(* PLC project MotionTest1, Higen MCL 1 *)
(* stored: creationDateTime 2012-01-06T15:20:13, modificationDateTime 2026-03-05T12:13:42 *)

FUNCTION_BLOCK BlendTest
  VAR
    moveA : MC_MoveAbsolute;
    switch : MC_Power;
    readpos : MC_ReadActualPosition;
    setpos : MC_SetPosition;
    Block1 : MC_MoveAbsolute;
    readspeed : MC_ReadParameter;
  END_VAR
  VAR_INPUT
    Axis : AXIS_REF;
    Enable : BOOL;
    BlendMode : MC_BUFFER_MODE;
  END_VAR
  VAR_OUTPUT
    Done : BOOL;
    Pn : LREAL;
    Vn : LREAL;
  END_VAR

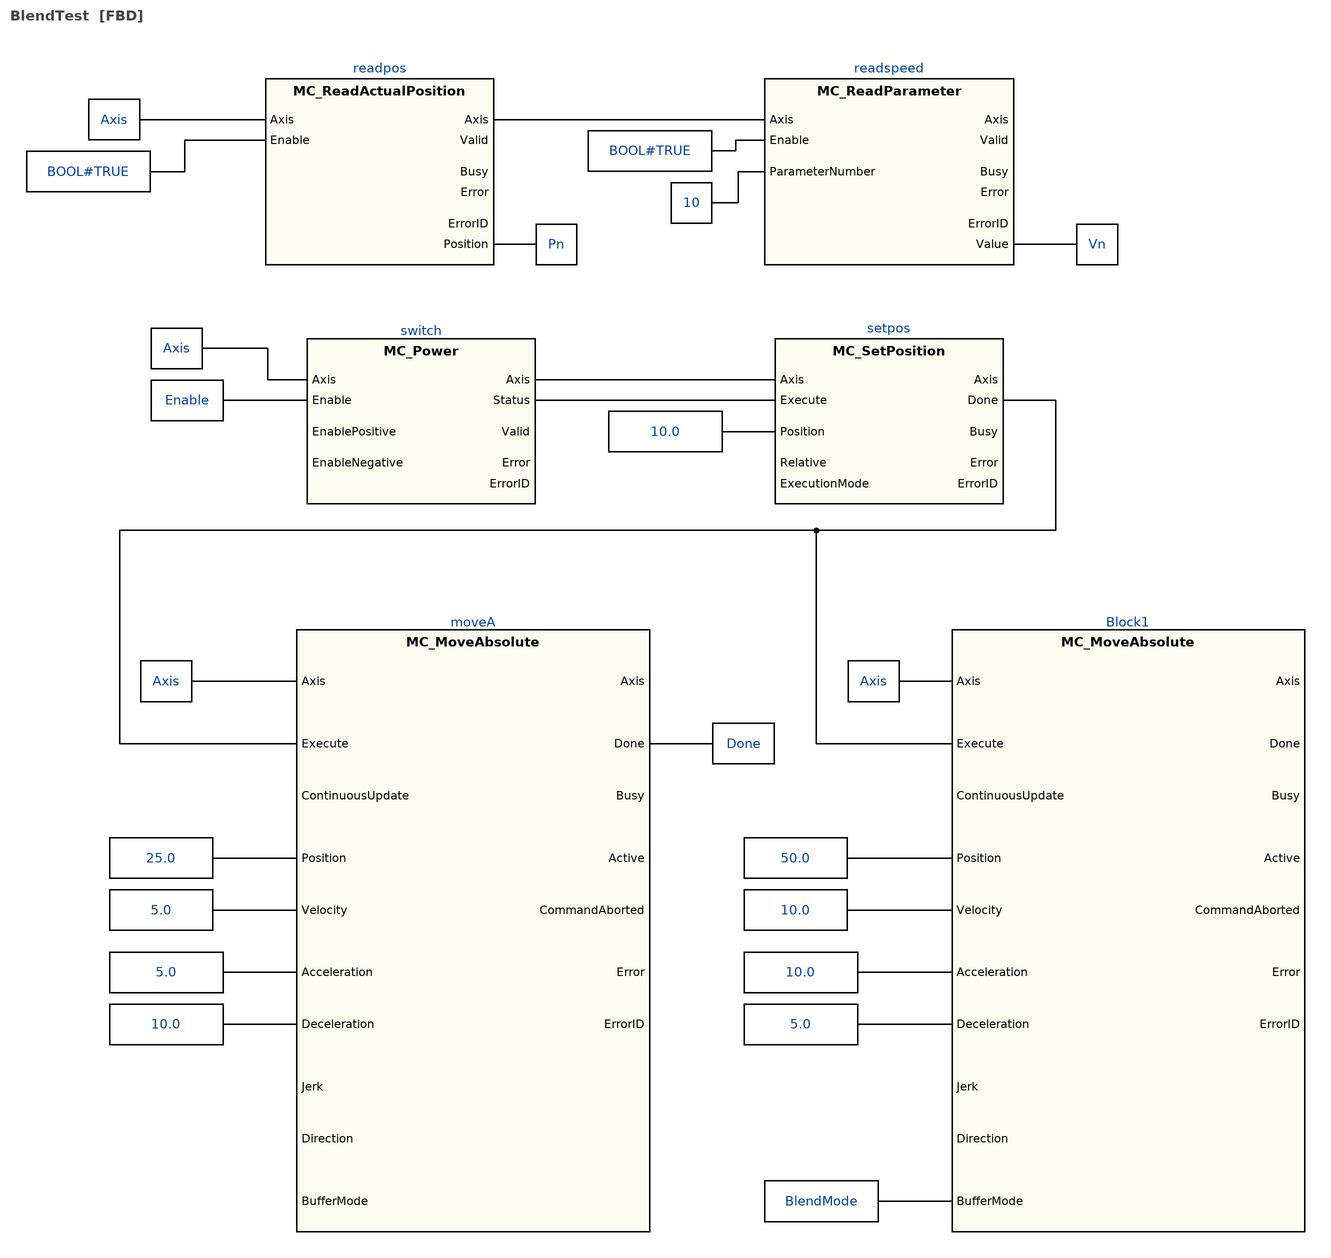
(* FBD diagram, written out as Structured Text *)
readpos(Axis := Axis, Enable := BOOL#TRUE);
Pn := readpos.Position;
switch(Axis := Axis, Enable := Enable);
setpos(Axis := switch.Axis, Execute := switch.Status, Position := 10.0);
moveA(Axis := Axis, Execute := setpos.Done, Position := 25.0, Velocity := 5.0, Acceleration := 5.0, Deceleration := 10.0);
Done := moveA.Done;
readspeed(Axis := readpos.Axis, Enable := BOOL#TRUE, ParameterNumber := 10);
Vn := readspeed.Value;
Block1(Axis := Axis, Execute := setpos.Done, Position := 50.0, Velocity := 10.0, Acceleration := 10.0, Deceleration := 5.0, BufferMode := BlendMode);
END_FUNCTION_BLOCK

PROGRAM main
  VAR
    clock : ULINT;
    High : BlendTest;
    Low : BlendTest;
    Previous : BlendTest;
    Next : BlendTest;
    r1 : R_TRIG;
    Block1 : R_TRIG;
    Block2 : R_TRIG;
    Block3 : R_TRIG;
    Block4 : BlendTest;
    Block5 : R_TRIG;
    sim0 : MC_Sim;
    sim1 : MC_Sim;
    sim2 : MC_Sim;
    sim3 : MC_Sim;
    sim4 : MC_Sim;
  END_VAR
  VAR  (* added by the conversion: wires and edge detectors of the diagram *)
    _SEL45_OUT : ANY;
    _SEL11_OUT : ANY;
    _SEL13_OUT : ANY;
    _SEL16_OUT : ANY;
    _SEL22_OUT : ANY;
  END_VAR

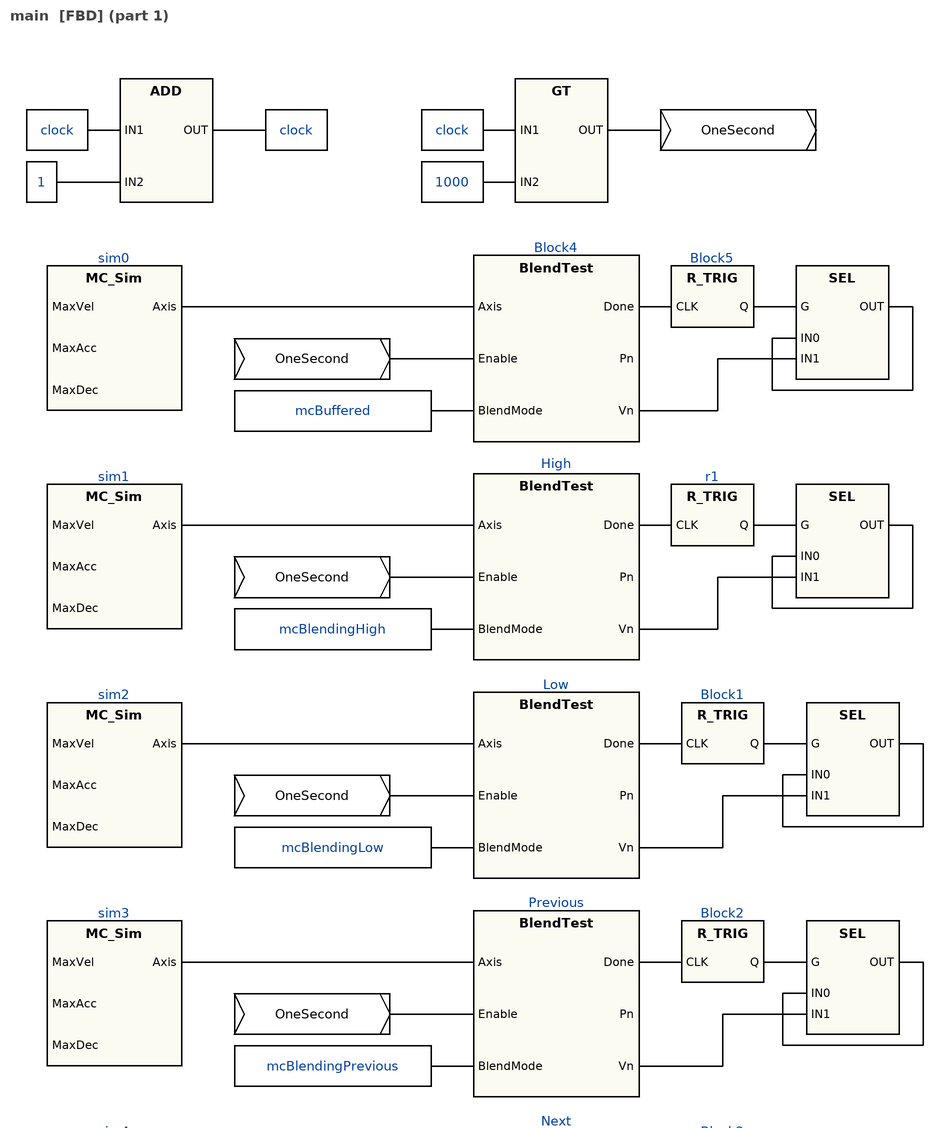
(* FBD diagram, written out as Structured Text *)
clock := clock + 1;
sim1();
High(Axis := sim1.Axis, Enable := clock > 1000, BlendMode := mcBlendingHigh);
sim2();
Low(Axis := sim2.Axis, Enable := clock > 1000, BlendMode := mcBlendingLow);
sim3();
Previous(Axis := sim3.Axis, Enable := clock > 1000, BlendMode := mcBlendingPrevious);
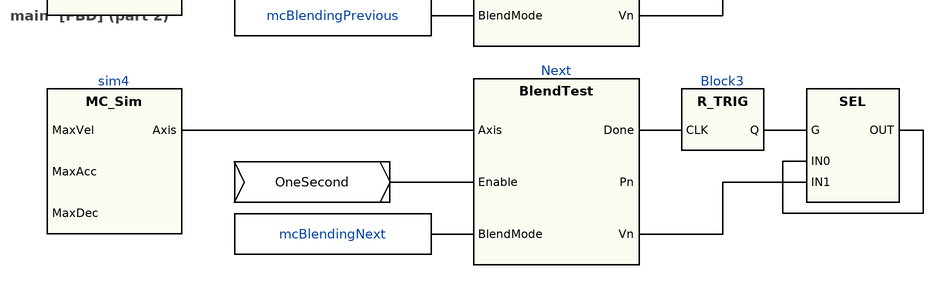
sim4();
Next(Axis := sim4.Axis, Enable := clock > 1000, BlendMode := mcBlendingNext);
r1(CLK := High.Done);
_SEL45_OUT := SEL(r1.Q, _SEL45_OUT, High.Vn);
Block1(CLK := Low.Done);
_SEL11_OUT := SEL(Block1.Q, _SEL11_OUT, Low.Vn);
Block2(CLK := Previous.Done);
_SEL13_OUT := SEL(Block2.Q, _SEL13_OUT, Previous.Vn);
Block3(CLK := Next.Done);
_SEL16_OUT := SEL(Block3.Q, _SEL16_OUT, Next.Vn);
sim0();
Block4(Axis := sim0.Axis, Enable := clock > 1000, BlendMode := mcBuffered);
Block5(CLK := Block4.Done);
_SEL22_OUT := SEL(Block5.Q, _SEL22_OUT, Block4.Vn);
END_PROGRAM

CONFIGURATION conf
  RESOURCE res ON PLC
    TASK milisecond(INTERVAL := T#1ms, PRIORITY := 0);
    PROGRAM maininstance WITH milisecond : main;
  END_RESOURCE
END_CONFIGURATION
